// TIA Portal project "Soru1" (V15)

(* hardware
DEVICE "S7-1200 station_1"  S7-1200 Station
   slot 0: "Rack_0"  S7-1200 Rack  Rack  V1.0
   slot 1: "PLC_1"  CPU 1214C DC/DC/DC  6ES7 214-1AG40-0XB0  V4.2
*)

// ===== PLC "PLC_1"  CPU 1214C DC/DC/DC =====

VAR_GLOBAL   // PLC tag table "Default tag table"
   "Durdur" AT %I0.0 : Bool;
   "Baslat" AT %I0.1 : Bool;
   "ÇıkısPMD" AT %Q0.0 : Bool;
END_VAR

// folder: System blocks/Program resources

DATA_BLOCK "IEC_Timer_0_DB"   // DB1
{ S7_Optimized_Access := 'TRUE' }
AUTHOR : Simatic
FAMILY : IEC
NAME : IEC_TMR
VERSION : 1.0
// stored: InstanceOfName IEC_TIMER
"IEC_TIMER"
BEGIN
END_DATA_BLOCK

DATA_BLOCK "IEC_Timer_0_DB_1"   // DB2
{ S7_Optimized_Access := 'TRUE' }
AUTHOR : Simatic
FAMILY : IEC
NAME : IEC_TMR
VERSION : 1.0
// stored: InstanceOfName IEC_TIMER
"IEC_TIMER"
BEGIN
END_DATA_BLOCK

// folder: (top level)

ORGANIZATION_BLOCK "Main"   // OB1, LAD, ProgramCycle
TITLE = "Main Program Sweep (Cycle)"
{ S7_Optimized_Access := 'TRUE' }
VERSION : 0.1
   VAR_INPUT
      Initial_Call : Bool;   // Initial call of this OB
      Remanence : Bool;   // =True, if remanent data are available
   END_VAR
BEGIN

REGION Network 1: Zaman Döngüsü
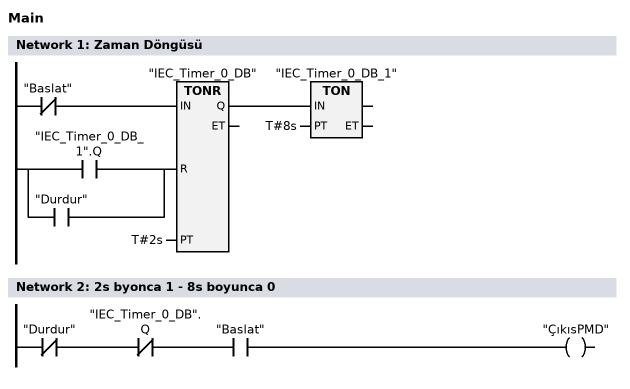
   "IEC_Timer_0_DB".TONR(IN := NOT "Baslat", R := "IEC_Timer_0_DB_1".Q OR "Durdur", PT := T#2s);
   "IEC_Timer_0_DB_1".TON(IN := "IEC_Timer_0_DB".Q, PT := T#8s);
END_REGION

REGION Network 2: 2s byonca 1 - 8s boyunca 0
   RUNG wire#powerrail
      I_Contact( "Durdur" )
      I_Contact( "IEC_Timer_0_DB".Q )
      Contact( "Baslat" )
      Coil( "ÇıkısPMD" )
   END_RUNG
   // the same network as SCL:
   "ÇıkısPMD" := NOT "Durdur" AND NOT "IEC_Timer_0_DB".Q AND "Baslat";
END_REGION
END_ORGANIZATION_BLOCK